// LS Electric XG5000 project: 유튜브방송용_2021082521
// PLC NewPLC

PROGRAM NewProgram (task: 스캔 프로그램)

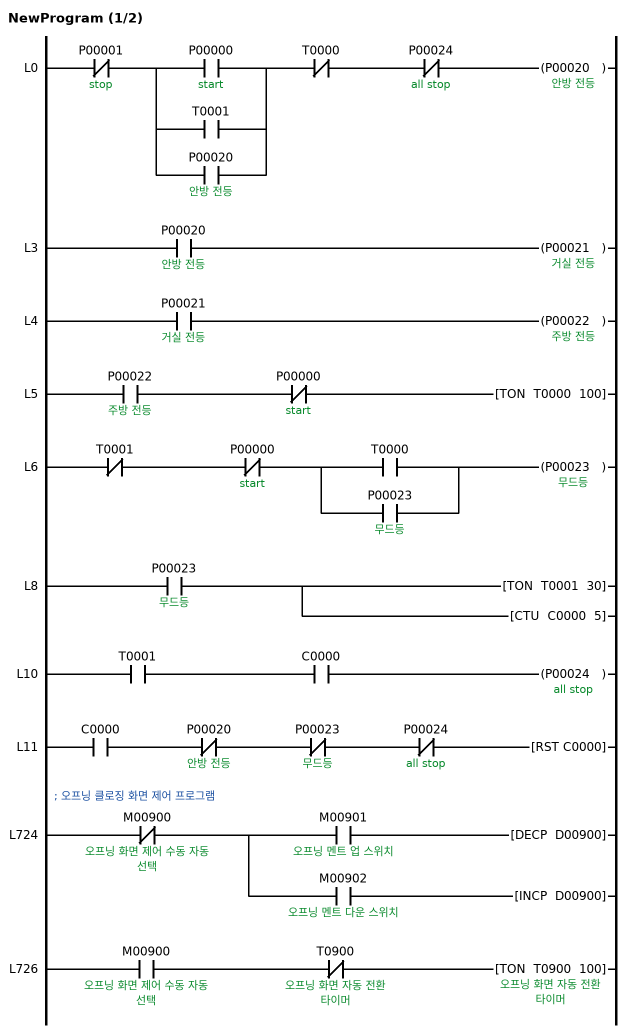
; L0
LOAD NOT  P00001	// stop
LOAD      P00000	// start
OR        T0001
OR        P00020	// 안방 전등
AND LOAD
AND NOT   T0000
AND NOT   P00024	// all stop
OUT       P00020	// 안방 전등
; L3
LOAD      P00020	// 안방 전등
OUT       P00021	// 거실 전등
; L4
LOAD      P00021	// 거실 전등
OUT       P00022	// 주방 전등
; L5
LOAD      P00022	// 주방 전등
AND NOT   P00000	// start
TON       T0000 100
; L6
LOAD NOT  T0001
AND NOT   P00000	// start
LOAD      T0000
OR        P00023	// 무드등
AND LOAD
OUT       P00023	// 무드등
; L8
LOAD      P00023	// 무드등
TON       T0001 30
CTU       C0000 5
; L10
LOAD      T0001
AND       C0000
OUT       P00024	// all stop
; L11
LOAD      C0000
AND NOT   P00020	// 안방 전등
AND NOT   P00023	// 무드등
AND NOT   P00024	// all stop
RST       C0000
// 오프닝 클로징 화면 제어 프로그램
; L724
LOAD NOT  M00900	// 오프닝 화면 제어 수동 자동 선택
MPUSH
AND       M00901	// 오프닝 멘트 업 스위치
DECP      D00900
MPOP
AND       M00902	// 오프닝 멘트 다운 스위치
INCP      D00900
; L726
LOAD      M00900	// 오프닝 화면 제어 수동 자동 선택
AND NOT   T0900	// 오프닝 화면 자동 전환 타이머
TON       T0900 100	// 오프닝 화면 자동 전환 타이머

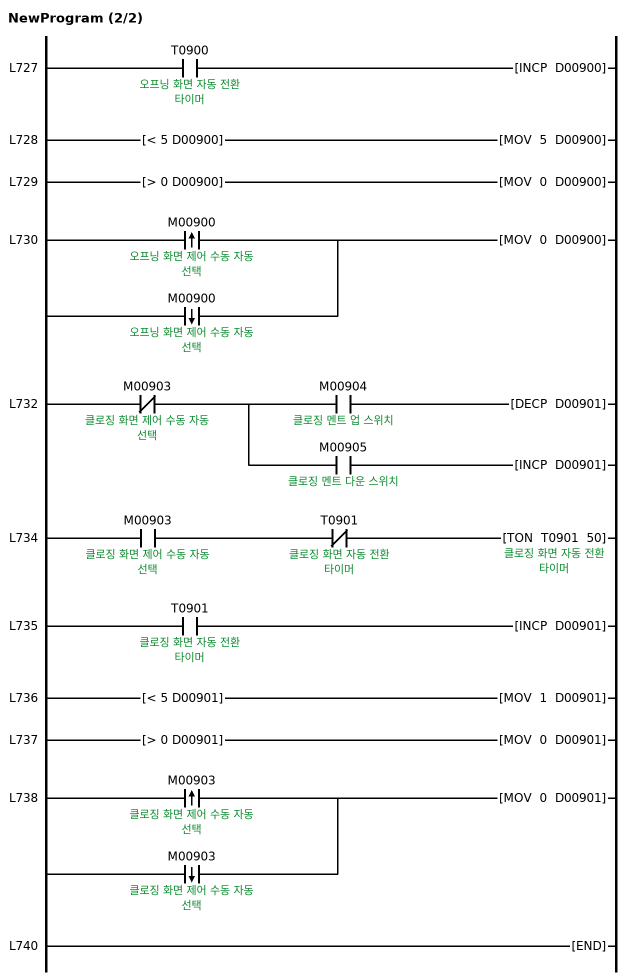
; L727
LOAD      T0900	// 오프닝 화면 자동 전환 타이머
INCP      D00900
; L728
LOAD<     5 D00900
MOV       5 D00900
; L729
LOAD>     0 D00900
MOV       0 D00900
; L730
LOADP     M00900	// 오프닝 화면 제어 수동 자동 선택
ORN       M00900	// 오프닝 화면 제어 수동 자동 선택
MOV       0 D00900
; L732
LOAD NOT  M00903	// 클로징 화면 제어 수동 자동 선택
MPUSH
AND       M00904	// 클로징 멘트 업 스위치
DECP      D00901
MPOP
AND       M00905	// 클로징 멘트 다운 스위치
INCP      D00901
; L734
LOAD      M00903	// 클로징 화면 제어 수동 자동 선택
AND NOT   T0901	// 클로징 화면 자동 전환 타이머
TON       T0901 50	// 클로징 화면 자동 전환 타이머
; L735
LOAD      T0901	// 클로징 화면 자동 전환 타이머
INCP      D00901
; L736
LOAD<     5 D00901
MOV       1 D00901
; L737
LOAD>     0 D00901
MOV       0 D00901
; L738
LOADP     M00903	// 클로징 화면 제어 수동 자동 선택
ORN       M00903	// 클로징 화면 제어 수동 자동 선택
MOV       0 D00901
; L740
END

VARIABLES AND COMMENTS (devices not used above)
P00002	BIT	주방 스위치